FUNCTION_BLOCK IMG_QUEUE_DELETE (* Basic FB with empty ECC *)
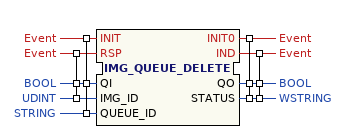
  EVENT_INPUT
    INIT WITH QI, QUEUE_ID;
    RSP WITH QI, IMG_ID;
  END_EVENT
  EVENT_OUTPUT
    INIT0 WITH QO, STATUS;
    IND WITH QO, STATUS;
  END_EVENT
  VAR_INPUT
    QI : BOOL;
    IMG_ID : UDINT;
    QUEUE_ID : STRING;
  END_VAR
  VAR_OUTPUT
    QO : BOOL;
    STATUS : WSTRING;
  END_VAR
END_FUNCTION_BLOCK
